ABB RobotStudio station: Project1_local_rebe.rspag

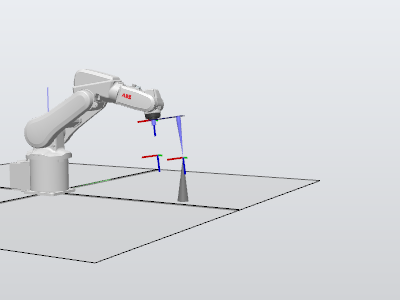
--- station ---
Station Project1_local_rebe (saved by RobotStudio 25.2.11220.0)
Controller Controlador1
  mechanical unit ROB_1: IRB120_3_58__01, 6 joints, base frame (0, 0, 0) mm
Layout (positions relative to the parent item):
  - IRB120_3_58__01 [mechanism, from %ABB.RobotStudio.Models.IRB120%\IRB120_3_58_G_01.rslib] at (0, 0, 0) mm; joint values [0.1358, 0.9791, -0.715, -0.0948, 1.1452, -0.0907] (rad or m)
  - Herramienta_piramidal [mechanism, from Components\Herramienta_piramidal.rslib] at (0, 0, 0) mm
  - Herramienta_de_soldadura [mechanism, from Components\Herramienta_de_soldadura.rslib] at (541.37, 67.68, 358.57) mm, rotated rx -173.88 ry 8.63 rz -164.72 deg
  - Pieza_1 [part] at (181.92, -13.18, 0) mm, size 50 x 49.2 x 200 mm
Attachment: Herramienta_de_soldadura is attached to IRB120_3_58__01 / Link6
Targets, tools, work objects and paths stored in the station and not in the controller backup, written as RAPID:
! task T_ROB1
MODULE CalibData
  PERS tooldata attach_cylinder:=[TRUE,[[0,0,0],[1,0,0,0]],[1,[-61.183,0.797,1],[1,0,0,0],0,0,0]];
  PERS tooldata puncture_figure:=[TRUE,[[-115.458,0.883,185],[1,0,0,0]],[1,[-61.183,0.797,1],[1,0,0,0],0,0,0]];
ENDMODULE


--- Controller Data/Controlador1/RAPID/TASK1/PROGMOD/CalibData.mod ---
MODULE CalibData
    PERS tooldata Herramienta_piramidal:=[TRUE,[[0,0,160],[1,0,0,0]],[0.2,[0,0,36.89],[1,0,0,0],0,0,0]];
ENDMODULE

--- Controller Data/Controlador1/RAPID/TASK1/PROGMOD/Module1.mod ---
MODULE Module1
	PERS tooldata Herramienta_piramidal_FP:=[TRUE,[[0,0,160],[1,0,0,0]],[0.2,[0,0,42.5],[1,0,0,0],0,0,0]];
	PERS tooldata Herramienta_de_soldadura:=[TRUE,[[0,0,184],[1,0,0,0]],[0.4,[0,0,42.5],[1,0,0,0],0,0,0]];
	TASK PERS wobjdata cone:=[FALSE,TRUE,"",[[0,0,0],[1,0,0,0]],[[0,0,0],[1,0,0,0]]];
    !***********************************************************
    !
    ! M?dulo:  Module1
    !
    ! Descripción:
    !   <Introduzca la descripción aquí>
    !
    ! Autor: r.castilla.2023
    !
    ! Versión: 1.0
    !
    !***********************************************************


    !***********************************************************
    !
    ! Procedimiento Main
    !
    !   Este es el punto de entrada de su programa
    !
    !***********************************************************
    PROC main()
        !Add your code here
    ENDPROC
ENDMODULE
